Fanuc KAREL source: kx00002.KL

-- PROVISIONAL review KL for V940-1; original PC SHA256 114b18af54f5b3e0be85f0568780c30eb291df9ec7b0e9e51f73a0b56262d760
-- Incomplete behavior may be omitted. Consult companion uncertainty JSON. Do not deploy.
PROGRAM KX00002
%NOLOCKGROUP
VAR
  I : INTEGER
  J : INTEGER
  B : BOOLEAN
  F : FILE
  S : STRING[80]
-- UNRESOLVED_DECL P type=000102
BEGIN
  -- V9_ZERO_TABLE_METADATA_HINT layout=0001; no indexed target words; source/name/runtime held
  -- UNRESOLVED_PC offsets 5-32; opcodes 22,3F,3F,3D
  -- UNRESOLVED_PC offsets 37-44; opcodes 22,39
  -- UNRESOLVED_PC offsets 49-53; opcodes 7F
END KX00002
